PROGRAM ModbusRead
VAR
	FB_MBReadInputs: FB_MBReadInputs;
	tReadInput: TON;
	bReadExecute: BOOL;
	
	IP 		: STRING:='127.0.0.1';
	Port 	: UINT:=505;
	ID 		: BYTE:=255;
	
	FB_MBReadInputRegs: FB_MBReadInputRegs;
	TON: TON;
	bInReg: BOOL;
END_VAR


tReadInput(IN:= NOT FB_MBReadInputs.bBusy, PT:=T#10MS , Q=>bReadExecute , ET=> );

FB_MBReadInputs(
	sIPAddr:= IP, 
	nTCPPort:= Port, 
	nUnitID:= ID, 
	nQuantity:= 16, 
	nMBAddr:= 0, 
	cbLength:= SIZEOF(InputBitArea), 
	pDestAddr:= ADR(InputBitArea), 
	bExecute:= bReadExecute, 
	tTimeout:= T#1S, 
	bBusy=> , 
	bError=> , 
	nErrId=> , 
	cbRead=> );

TON(IN:= NOT FB_MBReadInputRegs.bBusy , PT:=T#10MS , Q=>bInReg , ET=> );
	
FB_MBReadInputRegs(
	sIPAddr:= IP, 
	nTCPPort:= Port, 
	nUnitID:= ID, 
	nQuantity:= 3, 
	nMBAddr:= 0, 
	cbLength:= SIZEOF(InputWordArea), 
	pDestAddr:= ADR(InputWordArea), 
	bExecute:= bInReg, 
	tTimeout:= T#1S, 
	bBusy=> , 
	bError=> , 
	nErrId=> , 
	cbRead=> );

END_PROGRAM

(* stored: Version 1.1.0.1, ProductVersion 3.1.4024.6
   POU ModbusRead: Id {99c4169c-a3d5-4a25-ad98-775f18ef60f0}, SpecialFunc None *)
